// SIMATIC S7-200 project (STEP 7-Micro/WIN), CPU 224XP REL 02.01

SYMBOL_TABLE ANWENDER1
Ball_cnt_1       I0.2     // Ball verlässt Schraube 1
Ball_cnt_2       I0.3     // Ball verlässt Schraube 2
Ball_cnt_3       I0.4     // Ball verlässt Schraube 3
Air_ready        I0.5     // Pressure OK
Distr_top_rdy    I1.0     // Motor Verteiler oben BEREIT
Distr_bot_rdy    I1.1     // Motor Verteiler unten BEREIT
Pow_cnt_1        I1.2     // Power stroke bike 1
Pow_cnt_2        I1.3     // Power stroke bike 2
Pow_cnt_3        I1.4     // Power stroke bike 3
Cnt_disp_1       Q0.2     // Zähltakt Kopfdisplay 1
Blk_disp_1       Q0.3     // Blank Kopfdisplay 1 || Blank Upper Display 1
Rst_disp_1       Q0.4     // Reset Kopfdisplay 1
Cnt_disp_2       Q0.5     // Zähltakt Kopfdisplay 2 || Upper Count Display 2
Blk_disp_2       Q0.6     // Blank Kopfdisplay 2
Rst_disp_2       Q0.7     // Reset Kopfdisplay 2
Distr_top_en     Q1.0     // Enable Upper Motor
Distr_bot_en     Q1.1     // Enable Lower Motor
Cnt_disp_3       Q2.0     // Zähltakt Kopfdisplay 3
Blk_disp_3       Q2.1     // Blank Kopfdisplay 3
Rst_disp_3       Q2.2     // Reset Kopfdisplay 3
head_empty       Q2.4     // Crescendo
crescendo        Q2.5     // Ballentleerung Kopf
Vent_empt_1      Q2.6     // Ventil 3 in Display ohne Funktion
x1               Q2.7     // Ventil 4 in Display ohne Funktion
Note_1           Q3.0     // Ventil Note 1
Note_2           Q3.1     // Ventil Note 2
Note_3           Q3.2     // Ventil Note 3
Note_4           Q3.3     // Ventil Note 4
Note_5           Q3.4     // Ventil Note 5
Note_6           Q3.5     // Ventil Note 6
Note_7           Q3.6     // Ventil Note 7
Note_8           Q3.7     // Ventil Note 8
Note_cmpl        QB3      // Alle Noten im Ausgangsbyte
Ball_lift_en_1   Q4.0     // Turn on Steplifter and Screw 1
Ball_lift_en_2   Q4.1     // Turn on Steplifter and Screw 2
Ball_lift_en_3   Q4.2     // Turn on Steplifter and Screw 3
Disp_pow_cnt_1   Q4.4     // Zähltakt Leistungsdisplay 1
Disp_pow_cnt_2   Q4.5     // Zähltakt Leistungsdisplay 2
Disp_pow_mem     Q4.6     // Blank Leistungsdisplay 1+2
Disp_pow_rst     Q4.7     // Reset Leistungsdisplay 1+2
Wind_pow_in      AIW0     // Windleistung aus Strom berechnet
Distr_mot_1      AQW4     // Upper Distributor Motor Speed
Distr_mot_2      AQW6     // Lower Distributor Motor Speed
All_ready        M0.0     // Meets requirements for operation
Bike1_work       M0.1     // Someone Cycling on Bike 1
Bike2_work       M0.2     // Someone Cycling on Bike 2
Bike3_work       M0.3     // Someone Cycling on Bike 3
Music_play       M0.4     // Music is Playing
Cres_play        M0.5     // Crescendo runs
note_wrks        M0.6     // Schieberzeit 1 für Noten
hlp1_note_t      M0.7     // Hilfsmerker für M0.6
Flag_cresc       M1.0     // Crescendo Hubzylinder
time_tic_5ms     M2.0     // 4ms time symbols 1 cycle
Notes_all        MB3      // Byte für alle Noten
tic_5ms          T32      // 4ms Scores
Cnt_dis_up_1_t   T33      // Countimpuls für Display 1 oben
Cnt_dis_up_2_t   T34      // Countimpuls für Display 2 oben || Count pulse for upper display 2
Cnt_dis_up_3_t   T35      // Countimpuls für Display 3 oben
Note_next        T36      // Schrittzeit zur nächsten Auslesung
Cresc_delay      T38      // Wartezeit für Crescendoauslösung
Cresc_time       T39      // Ventilzeit Crescendo
Cresc_load       T40      // Ventilzeit Vorladen Crescendo
spr_up_time      T41      // Zeitverlängerung für Wischer oben
spr_bot_time     T42      // Zeitverlängerung für Wischer unten
Delay_music      T43      // Wartezeit bis Musik abspielen
Shot_time_1      T97      // Schieberzeit Töne 1
Shot_time_2      T98      // Schieberzeit Töne 2
note_time_1      T99      // Zeit zur nächsten Note
note_time_2      T100     // Zeit zur nächsten Note
Bike1_hold       T101     // Follow-up time Bike 1
Bike2_hold       T102     // Follow-up time Bike 2
Bike3_hold       T103     // Follow-up time Bike 3
Blk_disp_up_all  T104     // Alle oberen Display verzögert blanken || Upper Displays Blank
Rst_disp_up_all  T105     // Alle oberen Display verzögert rücksetzen
Rst_disp_bot_delay T106     // Wartezeit für Tastendruck Rücksetzen Displays Stele || Wait on key bot reset
Rst_disp_bot_en  T107     // Steuerzeit Displayreset Stele || Timing display reset bottom
Cnt_wind_time    T108     // Zählzeit Display Wind
Mem_wind_time    T109     // Memoryzeit Display Wind
Cnt_bike_time    T110     // Zählzeit Display Fahrräder
Mem_bike_time    T111     // Memoryzeit Display Fahrräder
note_mov_T1      T121     // Schieberzeit Note 1
note_mov_T2      T122     // Schieberzeit Note 2
note_mov_T3      T123     // Schieberzeit Note 3
note_mov_T4      T124     // Schieberzeit Note 4
note_mov_T5      T125     // Schieberzeit Note 5
note_mov_T6      T126     // Schieberzeit Note 6
note_mov_T7      T127     // Schieberzeit Note 7
note_mov_T8      T128     // Schieberzeit Note 8
note_run_1       T131     // Laufzeit Note 1
note_run_2       T132     // Laufzeit Note 2
note_run_3       T133     // Laufzeit Note 3
note_run_4       T134     // Laufzeit Note 4
note_run_5       T135     // Laufzeit Note 5
note_run_6       T136     // Laufzeit Note 6
note_run_7       T137     // Laufzeit Note 7
note_run_8       T138     // Laufzeit Note 8
Ball_numbers     VW0      // Number of balls moved by auger
Hit_number       VW2      // Auslösezahl für Musikspiel || Ball Counter Limit
Wind_pow_act     VD4      // Aktuelle Windleistung || Current wind power
Wind_pow_mem     VD8      // Gespeicherte Windleistung || Stored Wind Power
Bike_pow_act     VD12     // Aktuelle Fahrradleistung || Current bike Power
Bike_pow_mem     VD16     // Gespeicherte Fahrradleistung || Saved bike Power
Bike_tic_all     VD20     // Alle Fahrradticker || All Bike Values
Ball_nrs_1       VW30     // Number of balls bike 1
Ball_nrs_2       VW32     // Number of balls bike 2
Ball_nrs_3       VW34     // Number of balls bike 3
note_t_base      VW100    // Zeitbasis in ms
note_act_now     VB102    // aktuelle Note
note_steer       VB103    // Steuerbits
note_hlp_mem     VB104    // LB2 in [music] zwischenspeichern
wind_work_dif    VD108    // Momentane differentielle Leistung || Current Differential Power
wind_work_cum    VD112    // Kumulierte Leistung modulo 1kWh (3600000) || Cumulative performance  mod(1kWh)
Point_next_note  VD990    // Zeiger auf nächste Note
END_SYMBOL_TABLE

ORGANIZATION_BLOCK MAIN:OB1
TITLE=Test program for head [upper electronics] (digital displays, auger motor, tone valves, crescendo valves, drain)
// 
// E0.0, E0.1 Reserved
// E0.6, E0.7 Free
// E1.5 Free
// E2.0 bis E3.6 Free
// A0.0, A0.1 Reserved
// A2.3 Free
// A2.5 Spare valve [2]
// A2.6 Spare valve [3]
// 
// AEW2 Free
// AAW0 Free
// AAW2 Dummy (not important)
// 
BEGIN
Network 1
// Start up
?000                         //Startup routine.If the system is not yet presurized, wait.
?000                         //If the system is pressurized the system can start.
?000
LD     SM0.1                 // First Scan
ON     Air_ready:I0.5        // No Air Pressure
FILL   0, MW0, 16            // Clear all flags
LDN    SM0.1
A      Air_ready:I0.5        // Pressure
=      All_ready:M0.0        // The system is ready, it can begin other operations
?000
Network 2
// Times Clock
?000                         // Once the startup routine has completed and the system is pressurized
?000                         // Start and continue a clock signal on M2.0 at 200Hz
LD     All_ready:M0.0
AN     time_tic_5ms:M2.0
TON    tic_5ms:T32, 5        // x 1ms
LD     tic_5ms:T32
=      time_tic_5ms:M2.0     // every 5ms high cycle
Network 3
// Recognize Run Bike
LD     All_ready:M0.0        // System available
A      Air_ready:I0.5        // Air available
// UN     Music_play:M0.4
?000                         // UN     Cres_play:M0.5
?000
?000                         // Enable the step lifter and screw if system is started and pressurized
=      Ball_lift_en_1:Q4.0   // Relay for step lifter + screw
=      Ball_lift_en_2:Q4.1   // Relay for step lifter + screw
=      Ball_lift_en_3:Q4.2   // Relay for step lifter + screw
?000
?000                         // Bike 1
?000                         // I1.2-I1.4 are interrupts. If a state change occurs on the interrupt line and the system is in a ready state, begin a timer that checks
// if the bike has moved in the last 30s keep the bike enabled
 // if the bike has moved in the last 30s keep the bike enabled
LD     Pow_cnt_1:I1.2
EU
LD     Pow_cnt_1:I1.2
ED
OLD
A      All_ready:M0.0
TOF    Bike1_hold:T101, 300  // x 100ms
?000
LD     Bike1_hold:T101
=      Bike1_work:M0.1       // Bike is moved
?000
?000                         // Bike 2
LD     Pow_cnt_2:I1.3
EU
LD     Pow_cnt_2:I1.3
ED
OLD
A      All_ready:M0.0
TOF    Bike2_hold:T102, 300  // x 100ms
LD     Bike2_hold:T102
=      Bike2_work:M0.2       // Bike is moved
?000
?000                         // Bike 3
LD     Pow_cnt_3:I1.4
EU
LD     Pow_cnt_3:I1.4
ED
OLD
A      All_ready:M0.0
TOF    Bike3_hold:T103, 300  // x 100ms
LD     Bike3_hold:T103
=      Bike3_work:M0.3       // Bike is moved
Network 4
// Verteilermotoren || Distributor Motors
LD     All_ready:M0.0
MOVW   0, MW8                // ?delete ago?
?000                         // LD     Distr_top_rdy:I1.0          // Top distributor motor ready
?000                         // If any of the bikes is enabled or music is playing and the system is ready, keep the system alive for 100s more. 
?000
LD     Bike1_work:M0.1
O      Bike2_work:M0.2
O      Bike3_work:M0.3
O      Music_play:M0.4
ALD
?000                         // Translation of "Zeitverlängerung für Wischer unten" = "Time extension for wiper top"
?000
TOF    spr_up_time:T41, 1000 // x 100ms
LD     spr_up_time:T41
=      Distr_top_en:Q1.0
MOVB   SMB28, MB8
MOVB   0, MB9
SRW    MW8, 1                // /2
LD     All_ready:M0.0
MOVW   MW8, Distr_mot_1:AQW4
?000
?000                         // 
?000
LD     All_ready:M0.0
MOVW   0, MW8                // ?delete ago?
//LD     Distr_bot_rdy:I1.1          // Bottom distributor motor ready
LD     Bike1_work:M0.1
O      Bike2_work:M0.2
O      Bike3_work:M0.3
O      Music_play:M0.4
ALD
TOF    spr_bot_time:T42, 1000 // x 100ms
LD     spr_bot_time:T42
=      Distr_bot_en:Q1.1
MOVB   SMB29, MB8
MOVB   0, MB9
SRW    MW8, 1                // /2
LD     All_ready:M0.0
MOVW   MW8, Distr_mot_2:AQW6
Network 5
// Oberes Displays || Top Displays
// Ballzählung || Ball Count
?000
?000                         // When a ball leaves the screw and the system is ready and upper displays are not blank, it increments the ball counter for the screw
?000                         // as well as the overall ball counter
?000                         // There is a delay to prevent double counting of balls.
LD     All_ready:M0.0
A      Ball_cnt_1:I0.2       // Upper half screw
AN     Blk_disp_up_all:T104  // ??Pause??
EU
INCW   Ball_numbers:VW0
INCW   Ball_nrs_1:VW30       // increment bike 1 ball counter
TOF    Cnt_dis_up_1_t:T33, 5 // x 10ms
LD     Cnt_dis_up_1_t:T33
=      Cnt_disp_1:Q0.2
LD     All_ready:M0.0
A      Ball_cnt_2:I0.3       // Upper half screw
AN     Blk_disp_up_all:T104  // ??Pause??
EU
INCW   Ball_numbers:VW0
INCW   Ball_nrs_2:VW32       // increment bike 2 ball counter
TOF    Cnt_dis_up_2_t:T34, 5 // x 10ms
LD     Cnt_dis_up_2_t:T34
=      Cnt_disp_2:Q0.5
LD     All_ready:M0.0
A      Ball_cnt_3:I0.4       // Upper half screw
AN     Blk_disp_up_all:T104  // ??Pause??
EU
INCW   Ball_numbers:VW0
INCW   Ball_nrs_3:VW34       // increment bike 3 ball counter
TOF    Cnt_dis_up_3_t:T35, 5 // x 10ms
LD     Cnt_dis_up_3_t:T35
=      Cnt_disp_3:Q2.0
Network 6
// Obere Displays || Upper Displays
// Reset und Blinken || Reset and Blinking
?000
?000                         // Upper Display startup routine
LD     All_ready:M0.0
A      Music_play:M0.4
EU
TOF    Blk_disp_up_all:T104, 50 // x 100ms
LD     Blk_disp_up_all:T104  // Einfrierzeit
ED                           // abgelaufen ?
TOF    Rst_disp_up_all:T105, 10 // x 100ms
?000
?000                         // Flash the Upper displays 
LD     Blk_disp_up_all:T104  // Clear upper Displays
A      SM0.5                 // 1Hz Clock
=      Blk_disp_1:Q0.3
=      Blk_disp_2:Q0.6
=      Blk_disp_3:Q2.1
?000
?000                         //Reset the upper displays if a signal is received
LD     Rst_disp_up_all:T105  // Anzeige oben löschen
=      Rst_disp_1:Q0.4
=      Rst_disp_2:Q0.7
=      Rst_disp_3:Q2.2
Network 7
// Musikstückauslösung
// Noten spielen
?000                         // Play music when the balls reach the counter and reset the counters
?000                         // Also includes code for manual testing of music states       
?000
LDW>=  Ball_nrs_1:VW30, Hit_number:VW2 // Bälle Fahrrad 1 || Balls by Bike 1
OW>=   Ball_nrs_2:VW32, Hit_number:VW2 // Bälle Fahrrad 2
OW>=   Ball_nrs_3:VW34, Hit_number:VW2 // Bälle Fahrrad 3
?000                         // UW>    Ball_numbers:VW0, Hit_number:VW2 // Anzahl der Bälle für Musikstück
?000
EU                           // If any of the ball counters reach the counter
LD     I2.0                  // *** Testzwecke *** Handbetrieb ***
AN     Music_play:M0.4       // ***
EU                           // *** Spielauslösung
OLD
?000
?000                         //Reset the ball counters
MOVW   0, Ball_numbers:VW0   // Zähler löschen
MOVW   0, Ball_nrs_1:VW30
MOVW   0, Ball_nrs_2:VW32
MOVW   0, Ball_nrs_3:VW34
S      Music_play:M0.4, 1
=      M30.0                 // für UP music
TOF    Cresc_load:T40, 40    // x 100ms
LD     Cresc_load:T40        // Crescendo vorladen
O      I2.1                  // *** NUR für Testzwecke ( Handbetrieb )
=      head_empty:Q2.4       // Vorladeschieber  
?000
LD     All_ready:M0.0
AN     Music_play:M0.4       // kein Musikstück
AN     Cres_play:M0.5        // kein Crescendo
MOVB   0, Notes_all:MB3      // Noten leeren
R      note_wrks:M0.6, 2     // Notenmerker löschen
LD     Music_play:M0.4
?000
?000                         //     Call the music (SBR0 subroutine)
CALL   music:SBR0, 1, M30.0, Notes_all:MB3, Flag_cresc:M1.0
//            Stück Nr./Start/Note/Crescendo
LD     All_ready:M0.0
MOVB   Notes_all:MB3, Note_cmpl:QB3
A      Flag_cresc:M1.0
LD     I2.2                  // *** NUR für Testzwecke ( Handbetrieb )
OLD                          // ***
=      crescendo:Q2.5        // Crescendoschieber
LD     All_ready:M0.0
A      crescendo:Q2.5
ED
R      Music_play:M0.4, 2    // und Crescendo
Network 8
// Anzeige Stele
LD     SM0.0                 // Always on
?000
?000                         //Calls the subroutine power (SBR1)
CALL   power:SBR1, Wind_pow_in:AIW0, I2.7, M30.1, MB4
//                    Wind power / RESET / Fault / Displayanst.
LD     SM0.0                 // Always on
ANDB   2#11111000, MB4       // Relevante Bits ausmaskieren
ANDB   2#111, QB4            // Relevante Ausgänge vorlöschen
ORB    MB4, QB4              // Relevante Ausgänge setzen
END_ORGANIZATION_BLOCK

SUBROUTINE_BLOCK music:SBR0
TITLE=Spiel das Musikprogramm ab
VAR_INPUT
play_nr:BYTE;	// LB0 Stück Nr. X
Start_play:BOOL;	// L1.0 Start (1Zyklus high)
END_VAR
VAR_OUTPUT
Note_x:BYTE;	// LB2 Note c bis h
Cresc:BOOL;	// L3.0 Crescendo
END_VAR
VAR
Note_cnt:DWORD;	// LD4 Listennummer
Notes_all:WORD;	// LW8 Noten
wyw:WORD;	// LW10 Rubbelmerker
END_VAR
BEGIN
Network 1
// Vorab
// Lied 1 ab VW1000 ; 2 ab VW1200 ; 3 ab VW1400 ....
LD     #Start_play:L1.0
FILL   0, LW4, 7             // alles löschen
MOVB   0, #Note_x:LB2
MOVD   &VB1000, Point_next_note:VD990 // Zeiger 1. Lied Zeitbasis (Wort)
BTI    #play_nr:LB0, #wyw:LW10 // Lied Nr. wandeln 1
ITD    #wyw:LW10, #Note_cnt:LD4 // wandeln 2
-D     1, #Note_cnt:LD4
*D     200, #Note_cnt:LD4
+D     #Note_cnt:LD4, Point_next_note:VD990
MOVW   *Point_next_note:VD990, note_t_base:VW100 // Zeitbasis holen
/I     10, note_t_base:VW100 // für 10ms Timer vorbereiten
+D     2, Point_next_note:VD990 // Zeiger für erste Note (Byte)
TOF    Delay_music:T43, 10   // x 100ms
LD     Delay_music:T43
ED
S      note_wrks:M0.6, 1
MOVB   2#1, note_steer:VB103 // Steuerbit setzen
Network 2
// Note holen und sichern
LD     note_wrks:M0.6        // Musik spielt
AN     Cres_play:M0.5        // kein Crescendo
AN     hlp1_note_t:M0.7
TON    Note_next:T36, note_t_base:VW100 // x 10ms
LD     Note_next:T36
=      hlp1_note_t:M0.7      // Schritt
LD     note_wrks:M0.6        // Musik spielt
EU
O      hlp1_note_t:M0.7      // Schritt
LD     Cres_play:M0.5
ED
OLD
=      L11.0                 // tick
LD     L11.0                 // tick
AB=    note_steer:VB103, 2#1 // Steuerbit Musik
AN     Cres_play:M0.5
MOVW   *Point_next_note:VD990, #Notes_all:LW8 // Note holen
MOVB   LB9, note_act_now:VB102 // Noten sichern
MOVB   LB8, note_steer:VB103 // Steuerbits sichern
+D     2, Point_next_note:VD990 // Zeiger für nächste Note
LD     Music_play:M0.4
AB=    note_steer:VB103, 2#11 // Anforderung Crescendo
EU
S      Cres_play:M0.5, 1
LD     Cres_play:M0.5
TON    Cresc_delay:T38, 20   // x 100ms
LD     Cresc_delay:T38
EU
TOF    Cresc_time:T39, 50    // x 100ms
LD     Cresc_time:T39
=      #Cresc:L3.0
LD     note_wrks:M0.6
AB=    note_steer:VB103, 0   // keine Steuerbits
AB=    note_hlp_mem:VB104, 0 // keine Note(n) aktiv
AN     Cres_play:M0.5
R      Music_play:M0.4, 5    // alles AUS
JMP    41
Network 3
// Haste Töne ?
// Ton 1-4
LD     Music_play:M0.4
MOVB   note_act_now:VB102, LB9
MOVB   2#0, #Note_x:LB2
LD     L9.0                  // Anforderung Ton 1 [c]
EU
AN     note_run_1:T131       // Note nicht aktiv
TOF    note_mov_T1:T121, 4   // x 100ms
TOF    note_run_1:T131, 7    // x 100ms
LD     note_mov_T1:T121
=      L2.0                  // Schieber AUF Ton 1 [c]
LD     L9.1                  // Anforderung Ton 2 [d]
EU
AN     note_run_2:T132       // Note nicht aktiv
TOF    note_mov_T2:T122, 4   // x 100ms
TOF    note_run_2:T132, 7    // x 100ms
LD     note_mov_T2:T122
=      L2.1                  // Schieber AUF Ton 2 [d]
LD     L9.2                  // Anforderung Ton 3 [e]
EU
AN     note_run_3:T133       // Note nicht aktiv
TOF    note_mov_T3:T123, 4   // x 100ms
TOF    note_run_3:T133, 7    // x 100ms
LD     note_mov_T3:T123
=      L2.2                  // Schieber AUF Ton 3 [e]
LD     L9.3                  // Anforderung Ton 4 [f]
EU
AN     note_run_4:T134       // Note nicht aktiv
TOF    note_mov_T4:T124, 4   // x 100ms
TOF    note_run_4:T134, 7    // x 100ms
LD     note_mov_T4:T124
=      L2.3                  // Schieber AUF Ton 4 [f]
Network 4
// Haste Töne ?
// Ton 1-4
LD     L9.4                  // Anforderung Ton 5 [g]
EU
AN     note_run_5:T135       // Note nicht aktiv
TOF    note_mov_T5:T125, 4   // x 100ms
TOF    note_run_5:T135, 7    // x 100ms
LD     note_mov_T5:T125
=      L2.4                  // Schieber AUF Ton 5 [g]
LD     L9.5                  // Anforderung Ton 6 [a]
EU
AN     note_run_6:T136       // Note nicht aktiv
TOF    note_mov_T6:T126, 4   // x 100ms
TOF    note_run_6:T136, 7    // x 100ms
LD     note_mov_T6:T126
=      L2.5                  // Schieber AUF Ton 6 [a]
LD     L9.6                  // Anforderung Ton 7 [h]
EU
AN     note_run_7:T137       // Note nicht aktiv
TOF    note_mov_T7:T127, 4   // x 100ms
TOF    note_run_7:T137, 7    // x 100ms
LD     note_mov_T7:T127
=      L2.6                  // Schieber AUF Ton 7 [h]
LD     L9.7                  // Anforderung Ton 8 [c']
EU
AN     note_run_8:T138       // Note nicht aktiv
TOF    note_mov_T8:T128, 4   // x 100ms
TOF    note_run_8:T138, 7    // x 100ms
LD     note_mov_T8:T128
=      L2.7                  // Schieber AUF Ton 8 [c']
LD     Music_play:M0.4
MOVB   #Note_x:LB2, note_hlp_mem:VB104
LBL    41
END_SUBROUTINE_BLOCK

SUBROUTINE_BLOCK power:SBR1
TITLE=Ermittelt die Leistung in der Stele
VAR_INPUT
wind_pow_cur:WORD;	// LW0 Momentanstrom x3 || Intstantaneous current x3
disp_reset:BOOL;	// L2.0 Displayreset unten || Reset Lower Display
END_VAR
VAR_IN_OUT
wind_i_malfunc:BOOL;	// L2.1 Fehlfunktion Stromfühler Wind || Malfunction Sensor for Turbine
END_VAR
VAR_OUTPUT
disp_bot_all:BYTE;	// LB3 Steuerbits für Display unten || Control bits for display below
END_VAR
VAR
malfunc_wind:BOOL;	// L4.0 Störung Stromfühler || Current fault sensor
Hz_1s:BOOL;	// L4.1 1Hz Takt
kWh_wind_cnt:BOOL;	// L4.2 Wind 1kWh mehr
help_wind_1:DINT;	// LD5 Hilfszahl 1 Wind
help_wind_2:REAL;	// LD9 Hilfszahl 2 Wind
END_VAR
BEGIN
Network 1
// Synchroniesieren der Anzeige nach Neustart || Synchronizes the display after restart/reset  
// oder RESET !!Vorsicht!!
LD     SM0.0                 // Always on
ANDB   2#11111000, #disp_bot_all:LB3 // Bit 0-2 ignorieren
LD     SM0.1                 // First Scan
MOVD   Wind_pow_mem:VD8, Wind_pow_act:VD4
MOVD   Bike_pow_mem:VD16, Bike_pow_act:VD12
MOVD   0, wind_work_cum:VD112 // kumulierte Leistungen löschen
MOVD   0, Bike_tic_all:VD20
LD     #disp_reset:L2.0
TON    Rst_disp_bot_delay:T106, 50 // x 100ms
LD     Rst_disp_bot_delay:T106 // Resetverzögerung || Reset Delay
EU
TOF    Rst_disp_bot_en:T107, 4 // x 100ms
LD     Rst_disp_bot_en:T107
=      L3.7                  // Reset Lower Display 
MOVD   0, Wind_pow_act:VD4
MOVD   0, Wind_pow_mem:VD8
MOVD   0, Bike_pow_act:VD12
MOVD   0, Bike_pow_mem:VD16
MOVD   0, Bike_tic_all:VD20
MOVD   0, wind_work_cum:VD112
Network 2
// Windleistung ermitteln ; 4-20ma == 0-33A Ladestrom == 2-10V an AEW0(LW0) == 13107 - 65535
// Anzeige zeigt kWh
// 
// Determine wind power; 4-20ma == 0-33A  == 2-10V charging current to AIW0 (LW0) == 13107-65535
// Display shows kWh
LD     All_ready:M0.0
AW<    #wind_pow_cur:LW0, 5000
=      #malfunc_wind:L4.0    // Stromfühler defekt || Turbine malfunction detector
JMP    21
LD     All_ready:M0.0
ITD    #wind_pow_cur:LW0, #help_wind_1:LD5 // 16 -> 32 Bit
DTR    #help_wind_1:LD5, #help_wind_2:LD9 // 32 -> real
-R     6553.0, #help_wind_2:LD9 // Offset abziehen || Pull offset
/R     794.0, #help_wind_2:LD9 // normieren auf 33A (MAX) || Normalized to 33A (MAX)
*R     12.0, #help_wind_2:LD9 // x Batteriespannung (12V) = Watt || * 12V to get watts
ROUND  #help_wind_2:LD9, #help_wind_1:LD5 // real -> 32 Bit mit runden || Bit rounding
MOVD   #help_wind_1:LD5, wind_work_dif:VD108
AD<    wind_work_dif:VD108, 2 // Weniger 1W (Rauschen) || 1W is noise - Ignore
MOVD   0, wind_work_dif:VD108 // keine Ladung || No charge
LD     All_ready:M0.0
A      SM0.5                 // 1Hz Clock
EU
=      #Hz_1s:L4.1
+D     wind_work_dif:VD108, wind_work_cum:VD112 // Addieren zu kumulierter Leistung || Add to cumulative output
LDD>=  wind_work_cum:VD112, 3600000 // 1kWh
AN     Cnt_wind_time:T108    // Sicherheit
AN     Mem_wind_time:T109    // Sicherheit
-D     3600000, wind_work_cum:VD112 // abziehen
=      #kWh_wind_cnt:L4.2    // Anzeige Wind +1 Merker
LD     #kWh_wind_cnt:L4.2
TOF    Cnt_wind_time:T108, 4 // x 100ms
LD     Cnt_wind_time:T108
=      L3.4                  // cnt Display Wind +1
ED
INCD   Wind_pow_act:VD4      // + 1kWh
LD     L3.7                  // Reset
ED
OLD
TOF    Mem_wind_time:T109, 4 // x 100ms
LD     Mem_wind_time:T109
=      L3.6                  // Mem Display Wind
ED
MOVD   Wind_pow_act:VD4, Wind_pow_mem:VD8 // Memory sichern
LBL    21
Network 3
// Fahrradleistung ermitteln
// Teil 1: Leistungsimpulse einsammeln
// 
// 
LD     Pow_cnt_1:I1.2        // Fahrradticker 1
EU
INCD   Bike_tic_all:VD20     // Tickzähler gesamt
LD     Pow_cnt_1:I1.2
ED
INCD   Bike_tic_all:VD20
LD     Pow_cnt_2:I1.3        // Fahrradticker 2
EU
INCD   Bike_tic_all:VD20
LD     Pow_cnt_2:I1.3
ED
INCD   Bike_tic_all:VD20
LD     Pow_cnt_3:I1.4        // Fahrradticker 3
EU
INCD   Bike_tic_all:VD20
LD     Pow_cnt_3:I1.4
ED
INCD   Bike_tic_all:VD20
Network 4
// Fahrradleistung ermitteln
// Teil 2: Auswertung
// 
// Determine Bike Performance
// Part 2: Evaluation
?000
?000
LDD>=  Bike_tic_all:VD20, 90000 // == 1kWh
AN     Cnt_bike_time:T110    // Sicherheit
AN     Mem_bike_time:T111    // Sicherheit
-D     90000, Bike_tic_all:VD20 // modulo
INCD   Bike_pow_act:VD12
TOF    Cnt_bike_time:T110, 4 // x 100ms
LD     Cnt_bike_time:T110
=      L3.5                  // Display Bike 1+
ED
LD     L3.7                  // Reset
ED
OLD
TOF    Mem_bike_time:T111, 4 // x 100ms
LD     Mem_bike_time:T111
=      L3.3                  // Memory bike
ED
MOVD   Bike_pow_act:VD12, Bike_pow_mem:VD16 // Memory sichern
Network 5
// Störung
LD     #malfunc_wind:L4.0    // Störung Windleistung
A      SM0.5                 // 1Hz Clock
=      #wind_i_malfunc:L2.1  // Ausgabe || There is an issue
?000
END_SUBROUTINE_BLOCK

DATA_BLOCK_TAB ANWENDER1
BEGIN
// Werte für Leistungsanzeige
         Ball_numbers        // aktuell eingelochte Bälle
         Hit_number, 25      // Mindestanzahl für Lied
         Wind_pow_act        // aktuelle Windleistung
         Wind_pow_mem        // letzte gespeicherte Windleistung
         Bike_pow_act        // aktuelle Fahrradleistung
         Bike_pow_mem        // letzte gespeicherte Fahrradleistung
         Bike_tic_all        // Fahrradticks
         Ball_nrs_1          // Bälle Fahrrad 1
         Ball_nrs_2          // Bälle Fahrrad 2
         Ball_nrs_3          // Bälle Fahrrad 3
// Merkvariablenbereich
         note_t_base         // music: Zeitbasis für Noten
// kommt von 1.Stelle Lied /10 für 10ms-Timer
         note_act_now        // music: aktuelles Notenabbild
         note_steer          // Steuerbits
         wind_work_dif       // power: differentielle Leistung
         wind_work_cum       // power: Pow_wind_cum
// 
// Die Lieder werden ab Adresse vw1000, dann 1200, 1400 usw. abgelegt.
// 1.Wort ist die Zeitbasis für den Notentakt
// Das linke Byte sind Steuerbits
// LSB+0 == Lied läuft, LSB+1 == Crescendo
// Das rechte Byte ist die Note
// LSB+0 == c, LSB+1 == d, ..., LSB+7 == c'
// In VD990 wird der Zeiger für die nächste zu spielende Note abgelegt.
         Point_next_note     // Zeiger auf nächste Note (Default)
// Tonleiter
VW1000   350                 // Zeitbasis in ms für Noten holen
VW1002   2#100000001         // c
VW1004   2#100000010         // d
VW1006   2#100000100         // e
VW1008   2#100001000         // f
VW1010   2#100010000         // g
VW1012   2#100100000         // a
VW1014   2#101000000         // h
VW1016   2#110000000         // c'
VW1018   2#101000000         // h
VW1020   2#100100000         // a
VW1022   2#100010000         // g
VW1024   2#100001000         // f
VW1026   2#100000100         // e
VW1028   2#100000010         // d
VW1030   2#100000001         // c
VW1032   2#1100000000        // crescendo
VW1034   2#0                 // Ende
END_DATA_BLOCK_TAB
